// TIA Portal project "Lab5_Exp2_DrillingMachine" (V16)

(* hardware
DEVICE "S7300/ET200M station_1"  S7-300 station
   slot 0: "Rail_0"  Rail  6ES7 390-1***0-0AA0
   slot 2: "PLC_1"  CPU 317-2 PN/DP  6ES7 317-2EK14-0AB0  V3.2
      slot 2: "PROFINET interface_1"  PN-IO
         slot 1: "Port_1"  Port
         slot 2: "Port_2"  Port
*)

// ===== PLC "PLC_1"  CPU 317-2 PN/DP =====

VAR_GLOBAL   // PLC tag table "Default tag table"
   "diStartB" AT %I0.1 : Bool;
   "diClampPressure" AT %I0.3 : Bool;
   "diCarriageUp" AT %I0.4 : Bool;
   "diCarriageDown" AT %I0.5 : Bool;
   "doDrillMotor" AT %Q0.0 : Bool;
   "doCoolingPump" AT %Q0.1 : Bool;
   "doClampingDevice" AT %Q0.2 : Bool;
   "doLowerDrill" AT %Q0.3 : Bool;
   "tvDelayT1" AT %QW66 : Word;
   "tvDelayT2" AT %QW68 : Word;
   "mS_Stop" AT %M100.0 : Bool;
   "mS_MotorOn" AT %M100.1 : Bool;
   "mS_Clamp" AT %M100.2 : Bool;
   "mS_Coolant" AT %M100.4 : Bool;
   "mS_CarriageDown" AT %M100.5 : Bool;
   "mS_DelayT1" AT %M100.3 : Bool;
   "mT1Elapsed" AT %M101.0 : Bool;
   "mT2Elapsed" AT %M101.1 : Bool;
   "DelayT1" AT %T1 : Timer;
   "DelayT2" AT %T2 : Timer;
   "Tag_1" AT %M200.0 : Bool;
   "mS_CarriageUp" AT %M100.6 : Bool;
   "mS_Unclamp" AT %M100.7 : Bool;
   "diMotor" AT %I0.0 : Bool;
   "diCoolantPressure" AT %I0.2 : Bool;
END_VAR

ORGANIZATION_BLOCK "Main"   // OB1, LAD
TITLE = "Main Program Sweep (Cycle)"
{ S7_Optimized_Access := 'FALSE' }
VERSION : 0.1
   VAR_TEMP
      OB1_EV_CLASS : Byte;   // Bits 0-3 = 1 (Coming event), Bits 4-7 = 1 (Event class 1)
      OB1_SCAN_1 : Byte;   // 1 (Cold restart scan 1 of OB 1), 3 (Scan 2-n of OB 1)
      OB1_PRIORITY : Byte;   // Priority of OB Execution
      OB1_OB_NUMBR : Byte;   // 1 (Organization block 1, OB1)
      OB1_RESERVED_1 : Byte;   // Reserved for system
      OB1_RESERVED_2 : Byte;   // Reserved for system
      OB1_PREV_CYCLE : Int;   // Cycle time of previous OB1 scan (milliseconds)
      OB1_MIN_CYCLE : Int;   // Minimum cycle time of OB1 (milliseconds)
      OB1_MAX_CYCLE : Int;   // Maximum cycle time of OB1 (milliseconds)
      OB1_DATE_TIME : Date_And_Time;   // Date and time OB1 started
   END_VAR
   VAR_TEMP   // added for the SCL form of the ladder/FBD networks
      _w1 : Bool;
      _s5time1 : S5Time;
   END_VAR
BEGIN

REGION Network 1: Setting mS_Stop
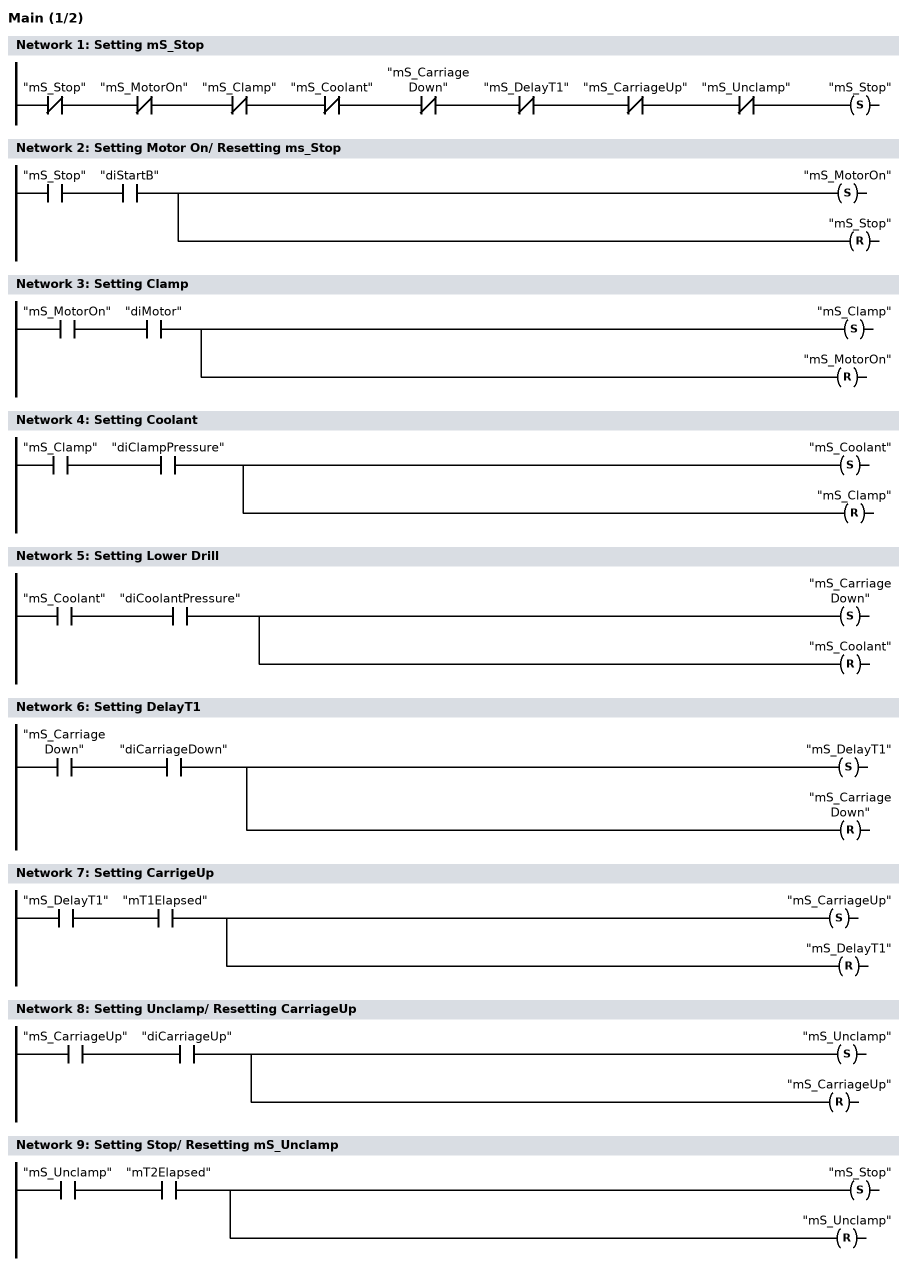
   RUNG wire#powerrail
      I_Contact( "mS_Stop" )
      I_Contact( "mS_MotorOn" )
      I_Contact( "mS_Clamp" )
      I_Contact( "mS_Coolant" )
      I_Contact( "mS_CarriageDown" )
      I_Contact( "mS_DelayT1" )
      I_Contact( "mS_CarriageUp" )
      I_Contact( "mS_Unclamp" )
      S_Coil( "mS_Stop" )
   END_RUNG
   // the same network as SCL:
   IF NOT "mS_Stop" AND NOT "mS_MotorOn" AND NOT "mS_Clamp" AND NOT "mS_Coolant" AND NOT "mS_CarriageDown" AND NOT "mS_DelayT1" AND NOT "mS_CarriageUp" AND NOT "mS_Unclamp" THEN
       "mS_Stop" := TRUE;
   END_IF;
END_REGION

REGION Network 2: Setting Motor On/ Resetting ms_Stop
   RUNG wire#powerrail
      Contact( "mS_Stop" )
      Contact( "diStartB" )
      wire#w1
      S_Coil( "mS_MotorOn" )
   END_RUNG
   RUNG wire#w1
      R_Coil( "mS_Stop" )
   END_RUNG
   // the same network as SCL:
   IF "mS_Stop" AND "diStartB" THEN
       "mS_MotorOn" := TRUE;
       "mS_Stop" := FALSE;
   END_IF;
END_REGION

REGION Network 3: Setting Clamp
   RUNG wire#powerrail
      Contact( "mS_MotorOn" )
      Contact( "diMotor" )
      wire#w1
      S_Coil( "mS_Clamp" )
   END_RUNG
   RUNG wire#w1
      R_Coil( "mS_MotorOn" )
   END_RUNG
   // the same network as SCL:
   IF "mS_MotorOn" AND "diMotor" THEN
       "mS_Clamp" := TRUE;
       "mS_MotorOn" := FALSE;
   END_IF;
END_REGION

REGION Network 4: Setting Coolant
   RUNG wire#powerrail
      Contact( "mS_Clamp" )
      Contact( "diClampPressure" )
      wire#w1
      S_Coil( "mS_Coolant" )
   END_RUNG
   RUNG wire#w1
      R_Coil( "mS_Clamp" )
   END_RUNG
   // the same network as SCL:
   IF "mS_Clamp" AND "diClampPressure" THEN
       "mS_Coolant" := TRUE;
       "mS_Clamp" := FALSE;
   END_IF;
END_REGION

REGION Network 5: Setting Lower Drill
   RUNG wire#powerrail
      Contact( "mS_Coolant" )
      Contact( "diCoolantPressure" )
      wire#w1
      S_Coil( "mS_CarriageDown" )
   END_RUNG
   RUNG wire#w1
      R_Coil( "mS_Coolant" )
   END_RUNG
   // the same network as SCL:
   IF "mS_Coolant" AND "diCoolantPressure" THEN
       "mS_CarriageDown" := TRUE;
       "mS_Coolant" := FALSE;
   END_IF;
END_REGION

REGION Network 6: Setting DelayT1
   RUNG wire#powerrail
      Contact( "mS_CarriageDown" )
      Contact( "diCarriageDown" )
      wire#w1
      S_Coil( "mS_DelayT1" )
   END_RUNG
   RUNG wire#w1
      R_Coil( "mS_CarriageDown" )
   END_RUNG
   // the same network as SCL:
   IF "mS_CarriageDown" AND "diCarriageDown" THEN
       "mS_DelayT1" := TRUE;
       "mS_CarriageDown" := FALSE;
   END_IF;
END_REGION

REGION Network 7: Setting CarrigeUp
   RUNG wire#powerrail
      Contact( "mS_DelayT1" )
      Contact( "mT1Elapsed" )
      wire#w1
      S_Coil( "mS_CarriageUp" )
   END_RUNG
   RUNG wire#w1
      R_Coil( "mS_DelayT1" )
   END_RUNG
   // the same network as SCL:
   IF "mS_DelayT1" AND "mT1Elapsed" THEN
       "mS_CarriageUp" := TRUE;
       "mS_DelayT1" := FALSE;
   END_IF;
END_REGION

REGION Network 8: Setting Unclamp/ Resetting CarriageUp
   RUNG wire#powerrail
      Contact( "mS_CarriageUp" )
      Contact( "diCarriageUp" )
      wire#w1
      S_Coil( "mS_Unclamp" )
   END_RUNG
   RUNG wire#w1
      R_Coil( "mS_CarriageUp" )
   END_RUNG
   // the same network as SCL:
   IF "mS_CarriageUp" AND "diCarriageUp" THEN
       "mS_Unclamp" := TRUE;
       "mS_CarriageUp" := FALSE;
   END_IF;
END_REGION

REGION Network 9: Setting Stop/ Resetting mS_Unclamp
   RUNG wire#powerrail
      Contact( "mS_Unclamp" )
      Contact( "mT2Elapsed" )
      wire#w1
      S_Coil( "mS_Stop" )
   END_RUNG
   RUNG wire#w1
      R_Coil( "mS_Unclamp" )
   END_RUNG
   // the same network as SCL:
   IF "mS_Unclamp" AND "mT2Elapsed" THEN
       "mS_Stop" := TRUE;
       "mS_Unclamp" := FALSE;
   END_IF;
END_REGION

REGION Network 10: Starting DelayT1
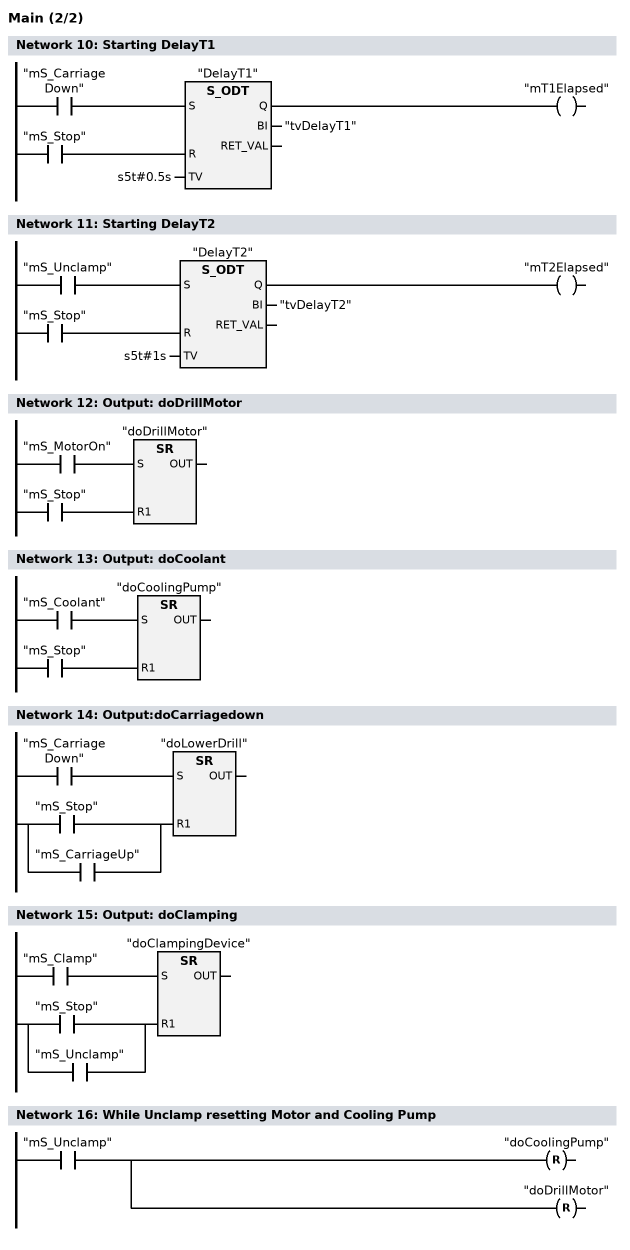
   RUNG wire#powerrail
      Contact( "mS_CarriageDown" )
      S_ODT(T_NO := "DelayT1", R := wire#w1, TV := s5t#0.5s, BI => "tvDelayT1", RET_VAL =>)
      Coil( "mT1Elapsed" )
   END_RUNG
   RUNG wire#powerrail
      Contact( "mS_Stop" )
   END_RUNG wire#w1
   // the same network as SCL:
   #_s5time1 := S_ODT(T_NO := "DelayT1",
                      S := "mS_CarriageDown",
                      R := "mS_Stop",
                      TV := s5t#0.5s,
                      Q => #_w1,
                      BI => "tvDelayT1");
   "mT1Elapsed" := #_w1;
END_REGION

REGION Network 11: Starting DelayT2
   RUNG wire#powerrail
      Contact( "mS_Unclamp" )
      S_ODT(T_NO := "DelayT2", R := wire#w1, TV := s5t#1s, BI => "tvDelayT2", RET_VAL =>)
      Coil( "mT2Elapsed" )
   END_RUNG
   RUNG wire#powerrail
      Contact( "mS_Stop" )
   END_RUNG wire#w1
   // the same network as SCL:
   #_s5time1 := S_ODT(T_NO := "DelayT2",
                      S := "mS_Unclamp",
                      R := "mS_Stop",
                      TV := s5t#1s,
                      Q => #_w1,
                      BI => "tvDelayT2");
   "mT2Elapsed" := #_w1;
END_REGION

REGION Network 12: Output: doDrillMotor
   RUNG wire#powerrail
      Contact( "mS_MotorOn" )
      S_SR(operand := "doDrillMotor", r1 := wire#w1)
   END_RUNG
   RUNG wire#powerrail
      Contact( "mS_Stop" )
   END_RUNG wire#w1
   // the same network as SCL:
   IF "mS_MotorOn" THEN
       "doDrillMotor" := TRUE;   // SR flip-flop
   END_IF;
   IF "mS_Stop" THEN "doDrillMotor" := FALSE; END_IF;
END_REGION

REGION Network 13: Output: doCoolant
   RUNG wire#powerrail
      Contact( "mS_Coolant" )
      S_SR(operand := "doCoolingPump", r1 := wire#w1)
   END_RUNG
   RUNG wire#powerrail
      Contact( "mS_Stop" )
   END_RUNG wire#w1
   // the same network as SCL:
   IF "mS_Coolant" THEN
       "doCoolingPump" := TRUE;   // SR flip-flop
   END_IF;
   IF "mS_Stop" THEN "doCoolingPump" := FALSE; END_IF;
END_REGION

REGION Network 14: Output:doCarriagedown
   RUNG wire#powerrail
      Contact( "mS_CarriageDown" )
      S_SR(operand := "doLowerDrill", r1 := wire#w1)
   END_RUNG
   RUNG wire#powerrail
      Contact( "mS_Stop" )
   END_RUNG wire#w1
   RUNG wire#powerrail
      Contact( "mS_CarriageUp" )
   END_RUNG wire#w1
   // the same network as SCL:
   IF "mS_CarriageDown" THEN
       "doLowerDrill" := TRUE;   // SR flip-flop
   END_IF;
   IF "mS_Stop" OR "mS_CarriageUp" THEN "doLowerDrill" := FALSE; END_IF;
END_REGION

REGION Network 15: Output: doClamping
   RUNG wire#powerrail
      Contact( "mS_Clamp" )
      S_SR(operand := "doClampingDevice", r1 := wire#w1)
   END_RUNG
   RUNG wire#powerrail
      Contact( "mS_Stop" )
   END_RUNG wire#w1
   RUNG wire#powerrail
      Contact( "mS_Unclamp" )
   END_RUNG wire#w1
   // the same network as SCL:
   IF "mS_Clamp" THEN
       "doClampingDevice" := TRUE;   // SR flip-flop
   END_IF;
   IF "mS_Stop" OR "mS_Unclamp" THEN "doClampingDevice" := FALSE; END_IF;
END_REGION

REGION Network 16: While Unclamp resetting Motor and Cooling Pump
   RUNG wire#powerrail
      Contact( "mS_Unclamp" )
      wire#w1
      R_Coil( "doCoolingPump" )
   END_RUNG
   RUNG wire#w1
      R_Coil( "doDrillMotor" )
   END_RUNG
   // the same network as SCL:
   IF "mS_Unclamp" THEN
       "doCoolingPump" := FALSE;
       "doDrillMotor" := FALSE;
   END_IF;
END_REGION
END_ORGANIZATION_BLOCK